FUNCTION_BLOCK FB_RC_Servo
VAR_INPUT
	stop : BOOL; // Stops motor at current position
	setpoint : INT; // Angle to reach
	rampSpeed : REAL; // Speed setpoint for servo angle
	trapezoidalProfileActive : BOOL; // Smooths speed of servo at start and end of movement
	servoAngleMin : INT; // Lower limit of function block output angle
	servoAngleMax : INT; // Upper limit of function block output angle
	rampCycleTime : TIME; // Set rampCycleTime to the same as the task sycle time
	rampStartPos : INT; // Starting position
END_VAR
VAR_OUTPUT
	currentPositionSetpoint : INT; // The actual output of function block
	error : STRING; // Error output for debug
END_VAR
VAR
	ramp : FB_CTRL_RAMP_GENERATOR;
	rampParameters : ST_CTRL_RAMP_GENERATOR_PARAMS;
END_VAR

rampParameters.fVeloNeg := rampSpeed;
rampParameters.fVeloPos := rampSpeed;
rampParameters.tCtrlCycleTime := rampCycleTime;
rampParameters.tTaskCycleTime := rampCycleTime;
ramp.fStart := rampStartPos;
ramp.fTarget := setpoint;

IF stop THEN
	ramp.bEnable := FALSE;
ELSE
	ramp.bEnable := TRUE;
END_IF

ramp(stParams := rampParameters);

END_FUNCTION_BLOCK

(* stored: Version 1.1.0.1, ProductVersion 3.1.4024.13
   POU FB_RC_Servo: Id {f9c2ce82-3d86-42bf-b049-c4e05cd4c773}, SpecialFunc None *)
